TYPE ST_INPUTS_LFT:
STRUCT


	stLinAct_POP1: 					ST_INPUTS_LinAct;
	stLinAct_POP2: 					ST_INPUTS_LinAct;
	stLinAct_POP3: 					ST_INPUTS_LinAct;
	
	stStaticConv_POP1:				ST_INPUTS_StaticConv;
	stStaticConv_POP2:				ST_INPUTS_StaticConv;
	stStaticConv_POP3:				ST_INPUTS_StaticConv;
	
	stTrayCentre_POP1:				ST_INPUTS_TrayCentre;
	stTrayCentre_POP2:				ST_INPUTS_TrayCentre;
	stTrayCentre_POP3:				ST_INPUTS_TrayCentre;
	
	stSequenceManager:				ST_INPUTS_SequenceManager_POP;
	
	
	stHandshakeUpstream:			ST_TrayExchangeHandshake;
	stHandshakeDownstream:			ST_TrayExchangeHandshake;
	
	bParamsInitialised: BOOL := FALSE;
	

END_STRUCT
END_TYPE

(* stored: Version 1.1.0.1, ProductVersion 3.1.4024.12
   DUT ST_INPUTS_LFT: Id {2ea78976-aff0-480c-a5c2-83bc5ce7f8a6} *)
